FUNCTION_BLOCK FB_RMatrix_Test EXTENDS FB_TestSuite
VAR_INPUT
END_VAR
VAR_OUTPUT
END_VAR
VAR
END_VAR

WhenSetFromAngleExpectResult();
WhenRotatedByIdentityExpectSame();
WhenRotatedTwiceExpectDouble();
WhenSetFrom321AnglesExpectResult();
WhenVectorRotatedExpectResult();
WhenReversedExpectOpposite();
WhenSetFromVectorsExpectResult();

METHOD PRIVATE WhenReversedExpectOpposite
VAR_INPUT
END_VAR
VAR
	R1 : RMatrix;
	R2 : RMatrix;
END_VAR
TEST('WhenReversedExpectOpposite');

// @TEST-RUN
R1.SetFromAngle(-PI/2,0);
R2.SetFromAngle(PI/2,0);
R2.Reverse();

// @TEST-ASSERT
AssertTrue(R2.IsEqual(R1),'Reversed R is not correct');

TEST_FINISHED();
END_METHOD

METHOD PRIVATE WhenRotatedByIdentityExpectSame
VAR_INPUT
END_VAR
VAR
	R1 : RMatrix;
	R2 : RMatrix;
END_VAR
TEST('WhenRotatedByIdentityExpectSame');

// @TEST-RUN
R1.RotateBy(R2);

// @TEST-ASSERT
AssertTrue(R1.IsEqual(R2),'Result is not the same');
AssertTrue(R2.GetDeterminant() = 1,'Determinant is not 1');

TEST_FINISHED();
END_METHOD

METHOD PRIVATE WhenRotatedTwiceExpectDouble
VAR_INPUT
END_VAR
VAR
	R1 : RMatrix;
	R2 : RMatrix;
	R3 : RMatrix;
END_VAR
TEST('WhenRotatedTwiceExpectDouble');

// @TEST-RUN
R1.SetFromAngle(PI/2,0);
R2.RotateBy(R1);
R2.RotateBy(R1);
R1.SetFromAngle(PI,0);
R3.RotateBy(R1);

// @TEST-ASSERT
AssertTrue(R3.IsEqual(R2),'Results are not identical');
AssertTrue(R2.GetRC(1,1) = -1,'Y Axis not reversed');
AssertTrue(R2.GetRC(2,2) = -1,'Z Axis not reversed');

TEST_FINISHED();
END_METHOD

METHOD PRIVATE WhenSetFrom321AnglesExpectResult
VAR_INPUT
END_VAR
VAR
	A1 : TaitBryanAngleOrientation;
	A2 : TaitBryanAngleOrientation;
	R1 : RMatrix;
	R2 : RMatrix;
	R3 : RMatrix;
END_VAR
TEST('WhenSetFrom321AnglesExpectResult');

// @TEST-RUN
A1.SetFromComponentsRad(PI/2,PI/2,PI/2,TaitBryanAngleSequence.ZYX);
R1 := A1.GetRMatrix();
R2.SetFromAngle(PI/2,0);
R3.RotateBy(R2);
R2.SetFromAngle(PI/2,1);
R3.RotateBy(R2);
R2.SetFromAngle(PI/2,2);
R3.RotateBy(R2);
A2 := R1.GetAngleSequence();

// @TEST-ASSERT
AssertTrue(R1.IsEqual(R3),'rotations from two methods are not equal');
AssertTrue(R1.GetRC(0,2) = 1,'R1 X vector not correct');
AssertTrue(R1.GetRC(1,1) = 1,'R1 Y vector not correct');
AssertTrue(R1.GetRC(2,0) = -1,'R1 Z vector not correct');
AssertTrue(R1.GetDeterminant() = 1,'R1 Determinant is not 1');

AssertTrue(R3.GetRC(0,2) = 1,'R3 X vector not correct');
AssertTrue(R3.GetRC(1,1) = 1,'R3 Y vector not correct');
AssertTrue(R3.GetRC(2,0) = -1,'R3 Z vector not correct');
AssertTrue(R3.GetDeterminant() = 1,'R3 Determinant is not 1');

TEST_FINISHED();
END_METHOD

METHOD PRIVATE WhenSetFromAngleExpectResult
VAR_INPUT
END_VAR
VAR
	R1 : RMatrix;
	R2 : RMatrix;
	R3 : RMatrix;
	R4 : RMatrix;
END_VAR
TEST('WhenSetFromAngleExpectResult');

// @TEST-RUN
R1.SetFromAngle(PI/2,0);
R2.SetFromAngle(PI/2,1);
R3.SetFromAngle(PI/2,2);
R4 := R3;
R3.Clear();

// @TEST-ASSERT
AssertTrue(R1.GetRC(0,0) = 1,'R1 X vector not correct');
AssertTrue(R1.GetRC(1,2) = -1,'R1 Y vector not correct');
AssertTrue(R1.GetRC(2,1) = 1,'R1 Z vector not correct');
AssertTrue(R1.GetDeterminant() = 1,'R1 Determinant is not 1');

AssertTrue(R2.GetRC(0,2) = 1,'R2 X vector not correct');
AssertTrue(R2.GetRC(1,1) = 1,'R2 Y vector not correct');
AssertTrue(R2.GetRC(2,0) = -1,'R2 Z vector not correct');
AssertTrue(R2.GetDeterminant() = 1,'R2 Determinant is not 1');

AssertTrue(R4.GetRC(0,1) = -1,'R4 X vector not correct');
AssertTrue(R4.GetRC(1,0) = 1,'R4 Y vector not correct');
AssertTrue(R4.GetRC(2,2) = 1,'R4 Z vector not correct');
AssertTrue(R4.GetDeterminant() = 1,'R4 Determinant is not 1');

TEST_FINISHED();
END_METHOD

METHOD PRIVATE WhenSetFromVectorsExpectResult
VAR_INPUT
END_VAR
VAR
	VX : Vector3;
	VY : Vector3;
	VZ : Vector3;
	R1 : RMatrix;
	RX : RMatrix;
	RY : RMatrix;
	RZ : RMatrix;
	RBad : RMatrix;
	
	ResX : BOOL;
	ResY : BOOL;
	ResZ : BOOL;
	ResBad : BOOL;
END_VAR
TEST('WhenSetFromVectorsExpectResult');

// @TEST-RUN
R1.SetFromAngle(PI/2,1);//90 deg rotation around Y
VX.SetFromComponents(0,0,-1);
VY.SetFromComponents(0,1,0);
VZ.SetFromComponents(1,0,0);
ResX := RX.SetFromVectorsYZ(VY,VZ);
ResY := RY.SetFromVectorsXZ(VX,VZ);
ResZ := RZ.SetFromVectorsXY(VX,VY);
ResBad := Rbad.SetFromVectorsXY(VX,VX);

// @TEST-ASSERT
AssertFalse(ResBad,'Parallel vectors should not have worked');
AssertTrue(ResX,'RX not calculated successfully');
AssertTrue(R1.IsNearlyEqual(RX,1E-9),'RX not calculated correctly');
AssertTrue(ResY,'RY not calculated successfully');
AssertTrue(R1.IsNearlyEqual(RY,1E-9),'RY not calculated correctly');
AssertTrue(ResZ,'RZ not calculated successfully');
AssertTrue(R1.IsNearlyEqual(RZ,1E-9),'RZ not calculated correctly');

TEST_FINISHED();
END_METHOD

METHOD PRIVATE WhenVectorRotatedExpectResult
VAR_INPUT
END_VAR
VAR
	R1 : RMatrix;
	V1 : Vector3;
	V2 : Vector3;
END_VAR
TEST('WhenVectorRotatedExpectResult');

// @TEST-RUN
R1.SetFromAngle(PI/2,1);
V1.X := 1;
V2 := R1.GetRotatedVector3(V1);

// @TEST-ASSERT
AssertTrue(V2.Z = -1,'Result is not in correct direction');
AssertTrue(V2.GetVectorMagnitude() = 1,'magnitude is not 1');

TEST_FINISHED();
END_METHOD

END_FUNCTION_BLOCK

(* stored: Version 1.1.0.1, ProductVersion 3.1.4024.9
   POU FB_RMatrix_Test: Id {29776a3c-62a7-4a52-9285-714d234bd6c2}, SpecialFunc None
   Method WhenReversedExpectOpposite: Id {e47eb044-1085-4952-9808-e96e8cc7d353}
   Method WhenRotatedByIdentityExpectSame: Id {cefa467e-239c-44b5-9555-39c6f4209af6}
   Method WhenRotatedTwiceExpectDouble: Id {da191774-0fa7-4b17-8fa8-29bdac82bc08}
   Method WhenSetFrom321AnglesExpectResult: Id {41d63c5a-9d95-43f4-a307-47376ec46b64}
   Method WhenSetFromAngleExpectResult: Id {565445fa-2ab3-4e2a-a94b-9dcc4ab7c985}
   Method WhenSetFromVectorsExpectResult: Id {7da436ae-ed2e-0f8f-030a-9a2316b96d5e}
   Method WhenVectorRotatedExpectResult: Id {ff1fca85-5a1f-458e-a62f-35a7e11201fe} *)
